Staubli VAL3: scroll.pgx

public program scroll(num x_nX, num x_nY, num x_nDim, num x_nPos)
// create a scroll bar
  local string l_sMessage
  local string l_sLine
  local num l_nPos
  local string l_sScrool
begin
  // use the scroll
  if x_nPos>0 and x_nPos<=100
    l_nPos=round(x_nDim*x_nPos/100)
    if l_nPos>0
      // make the scroll
      call strfill(l_sScrool,l_nPos,l_sScrool)
      call strfillchr(l_sScrool,l_sScrool,"■")
    endIf
    // make the line
    call strfill(l_sLine,x_nDim-l_nPos,l_sLine)
    call strfillchr(l_sLine,l_sLine,"─")
    l_sMessage="├"+l_sScrool+l_sLine+"┤"
    // show the line
    call type(x_nX,x_nY,l_sMessage)
  endIf
end
